{attribute 'qualified_only'}
VAR_GLOBAL
	dataman200_1 : TcoDatamanIO_v_5_x_x;
	dataman200_2 : TcoDatamanIO_v_5_x_x;
END_VAR

(* stored: Version 1.1.0.1, ProductVersion 3.1.4024.11
   GVL IO: Id {c261a2fb-3c28-068a-01a6-595efe5a78fd} *)
